{attribute 'linkalways'} 
{attribute 'no_explicit_call' := 'This FB is a CLASS and must be accessed using methods or properties'}
{attribute 'enable_dynamic_creation'}
FUNCTION_BLOCK Node_F_VN_MedianElementElementwise_INT EXTENDS VisionNode
VAR
    ipContainer : _ITcVnContainer;
    nMedian : _INT(0);
    hrPrev : _HRESULT(S_OK);
    hresult : _HRESULT(S_OK);
END_VAR

METHOD PUBLIC  Clone : I_Node
VAR
	pNode : POINTER TO Node_F_VN_MedianElementElementwise_INT;
END_VAR
pNode := __NEW(Node_F_VN_MedianElementElementwise_INT);
Clone := pNode^;
END_METHOD

METHOD FB_init : BOOL
VAR_INPUT
	bInitRetains : BOOL; // if TRUE, the retain variables are initialized (warm start / cold start)
	bInCopyCode : BOOL;  // if TRUE, the instance afterwards gets moved into the copy code (online change)
END_VAR
AddInput('ipContainer', ipContainer);
AddInput('nMedian', nMedian);
AddInput('hrPrev', hrPrev);
AddOutput('ipContainer', ipContainer);
AddOutput('hresult',hresult);
END_METHOD

METHOD PROTECTED OnExecute : HRESULT
hresult.Value := F_VN_MedianElementElementwise_INT(
    ipContainer := ipContainer.Value,
    nMedian := nMedian.Value,
    hrPrev:= hrPrev.Value);
END_METHOD

METHOD PUBLIC PreExecutionCheck
VAR_INPUT
	Check : I_PreExecutionChecks;
END_VAR
Check.IsTrue(ipContainer.IsValid, 'ipContainer must be a valid container');
END_METHOD

END_FUNCTION_BLOCK

(* stored: Version 1.1.0.1, ProductVersion 3.1.4024.13
   POU Node_F_VN_MedianElementElementwise_INT: Id {21919fa0-140c-4c06-976c-ee07c33aa1b7}, SpecialFunc None
   Folder Constructor: Id {55bfa021-99db-4043-809d-59d1bf5e1eb1}
   Method Clone: Id {667ca661-3928-43e0-833f-c0a4759c5894}
   Method FB_init: Id {9934a538-23aa-4bc6-aa90-3c8940c507e8}
   Method OnExecute: Id {c239996d-20d9-42ec-a91e-0184192aff84}
   Method PreExecutionCheck: Id {6162767c-1071-4ace-bc39-cad77bb8b2b3} *)
